// TIA Portal V20 export
TYPE "LER_typeVisionGapData"
// stored: Access Published
   STRUCT
      OK : Bool;
      NG : Bool;
      Complete : Bool;
      RnR1OK : Bool;
      RnR1NG : Bool;
      RnR1Complete : Bool;
      RnR3OK : Bool;
      RnR3NG : Bool;
      RnR3Complete : Bool;
      Data : "LER_typeVisionGapResultData";
   END_STRUCT;
END_TYPE
